TYPE TFMachinePalletizer_Layer_OLD :
STRUCT
	X			: REAL	:= 0.0;	(* READ	- (mm) Dimensione X *)
	Y			: REAL	:= 0.0;	(* READ	- (mm) Dimensione Y *)
	Z			: REAL	:= 0.0;	(* READ	- (mm) Dimensione Z *)
END_STRUCT
END_TYPE

(* stored: Version 1.1.0.1, ProductVersion 3.1.4024.11
   DUT TFMachinePalletizer_Layer_OLD: Id {8e418878-10a0-4173-a2a1-d3bd9d18dd70} *)
